(* Logix 5000 project; controller DUNEW2PLC1 vendor 1 type 14 code 221 rev 33.11; software revision 33.00; part 4 of 7 *)
(* tags used below, declared in another part *)
   BOOLS : BOOL[1024];
   DINTS : DINT[1024];
   idx_0 : DINT;
   idx_1 : DINT;
   idx_2 : DINT;
   REALS : REAL[1024];
   HomeTrigger : BOOL;
   MORE_STATS_S : BOOL[32];
   resetPB_S : BOOL;
   Safety_System_Healthy : BOOL;
   Safety_Tripped_S : BOOL;
   SegQueue : MotionSeg[32];
   X_Axis_SFX : SAFETY_FEEDBACK_INTERFACE;
   X_Axis_SLS : SAFELY_LIMITED_SPEED;
(* queued_motion, continued *)

ROUTINE MaxAbsCosSweep   (* ladder *)
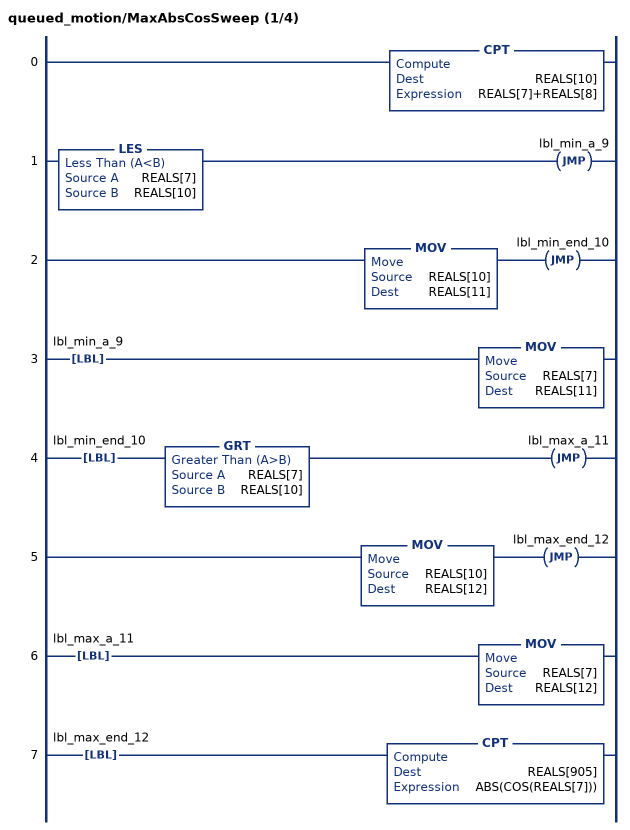
   0: CPT(REALS[10],REALS[7]+REALS[8]);
   1: LES(REALS[7],REALS[10])JMP(lbl_min_a_9);
   2: MOV(REALS[10],REALS[11])JMP(lbl_min_end_10);
   3: LBL(lbl_min_a_9)MOV(REALS[7],REALS[11]);
   4: LBL(lbl_min_end_10)GRT(REALS[7],REALS[10])JMP(lbl_max_a_11);
   5: MOV(REALS[10],REALS[12])JMP(lbl_max_end_12);
   6: LBL(lbl_max_a_11)MOV(REALS[7],REALS[12]);
   7: LBL(lbl_max_end_12)CPT(REALS[905],ABS(COS(REALS[7])));
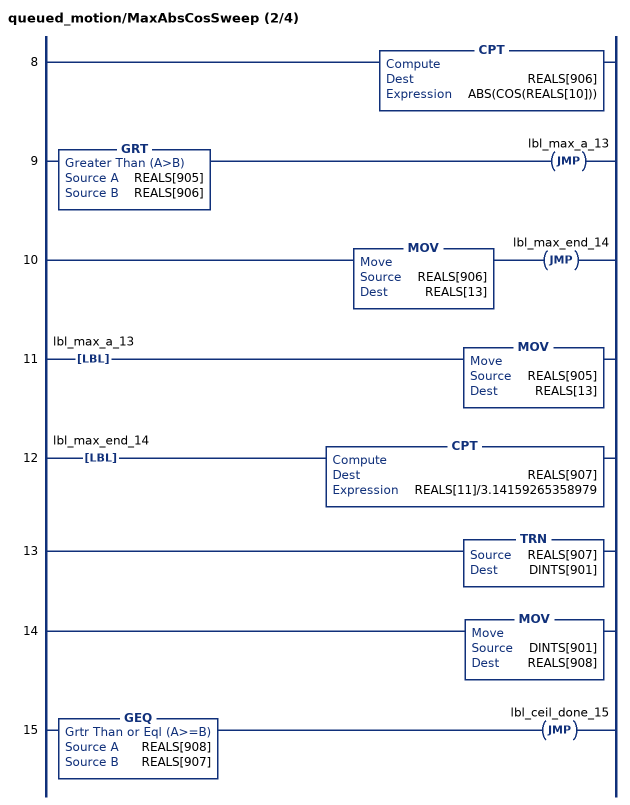
   8: CPT(REALS[906],ABS(COS(REALS[10])));
   9: GRT(REALS[905],REALS[906])JMP(lbl_max_a_13);
   10: MOV(REALS[906],REALS[13])JMP(lbl_max_end_14);
   11: LBL(lbl_max_a_13)MOV(REALS[905],REALS[13]);
   12: LBL(lbl_max_end_14)CPT(REALS[907],REALS[11]/3.14159265358979);
   13: TRN(REALS[907],DINTS[901]);
   14: MOV(DINTS[901],REALS[908]);
   15: GEQ(REALS[908],REALS[907])JMP(lbl_ceil_done_15);
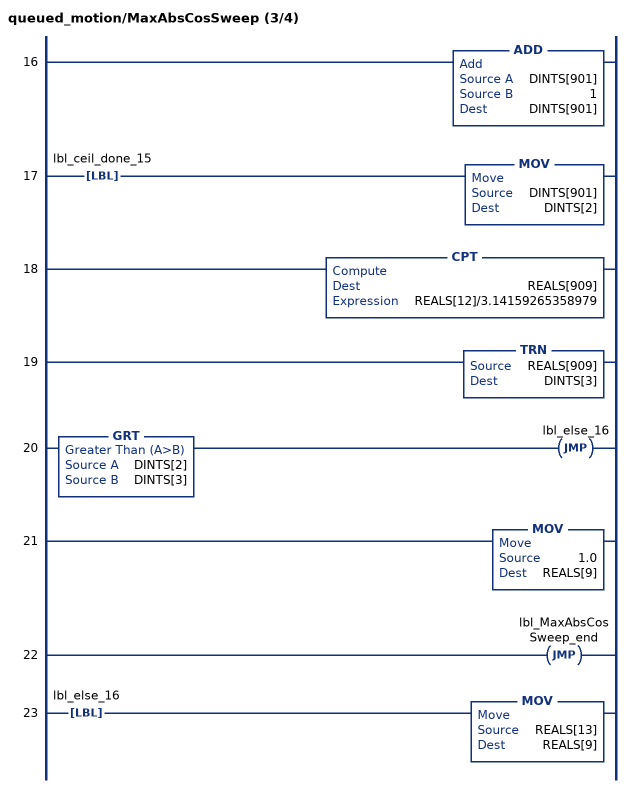
   16: ADD(DINTS[901],1,DINTS[901]);
   17: LBL(lbl_ceil_done_15)MOV(DINTS[901],DINTS[2]);
   18: CPT(REALS[909],REALS[12]/3.14159265358979);
   19: TRN(REALS[909],DINTS[3]);
   20: GRT(DINTS[2],DINTS[3])JMP(lbl_else_16);
   21: MOV(1.0,REALS[9]);
   22: JMP(lbl_MaxAbsCosSweep_end);
   23: LBL(lbl_else_16)MOV(REALS[13],REALS[9]);
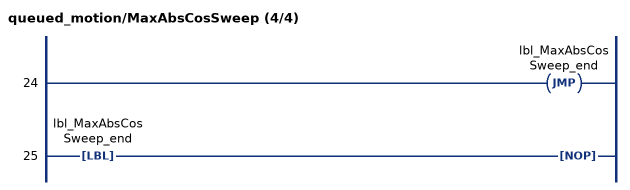
   24: JMP(lbl_MaxAbsCosSweep_end);
   25: LBL(lbl_MaxAbsCosSweep_end)NOP();
END_ROUTINE

ROUTINE MaxAbsSinSweep   (* ladder *)
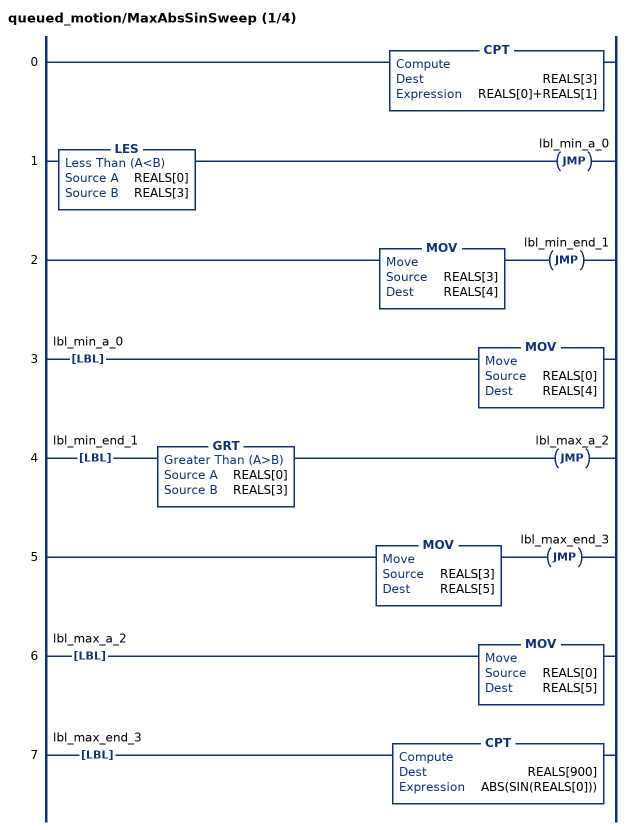
   0: CPT(REALS[3],REALS[0]+REALS[1]);
   1: LES(REALS[0],REALS[3])JMP(lbl_min_a_0);
   2: MOV(REALS[3],REALS[4])JMP(lbl_min_end_1);
   3: LBL(lbl_min_a_0)MOV(REALS[0],REALS[4]);
   4: LBL(lbl_min_end_1)GRT(REALS[0],REALS[3])JMP(lbl_max_a_2);
   5: MOV(REALS[3],REALS[5])JMP(lbl_max_end_3);
   6: LBL(lbl_max_a_2)MOV(REALS[0],REALS[5]);
   7: LBL(lbl_max_end_3)CPT(REALS[900],ABS(SIN(REALS[0])));
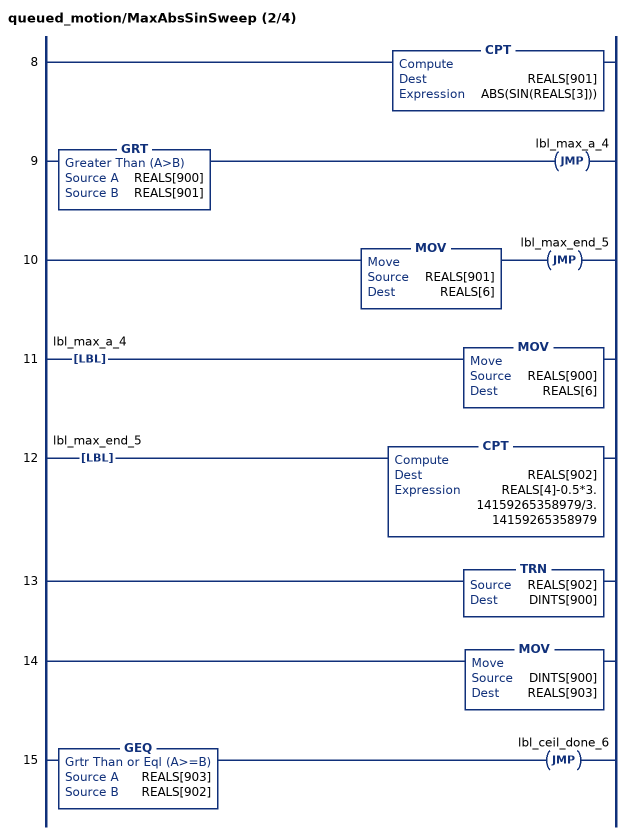
   8: CPT(REALS[901],ABS(SIN(REALS[3])));
   9: GRT(REALS[900],REALS[901])JMP(lbl_max_a_4);
   10: MOV(REALS[901],REALS[6])JMP(lbl_max_end_5);
   11: LBL(lbl_max_a_4)MOV(REALS[900],REALS[6]);
   12: LBL(lbl_max_end_5)CPT(REALS[902],REALS[4]-0.5*3.14159265358979/3.14159265358979);
   13: TRN(REALS[902],DINTS[900]);
   14: MOV(DINTS[900],REALS[903]);
   15: GEQ(REALS[903],REALS[902])JMP(lbl_ceil_done_6);
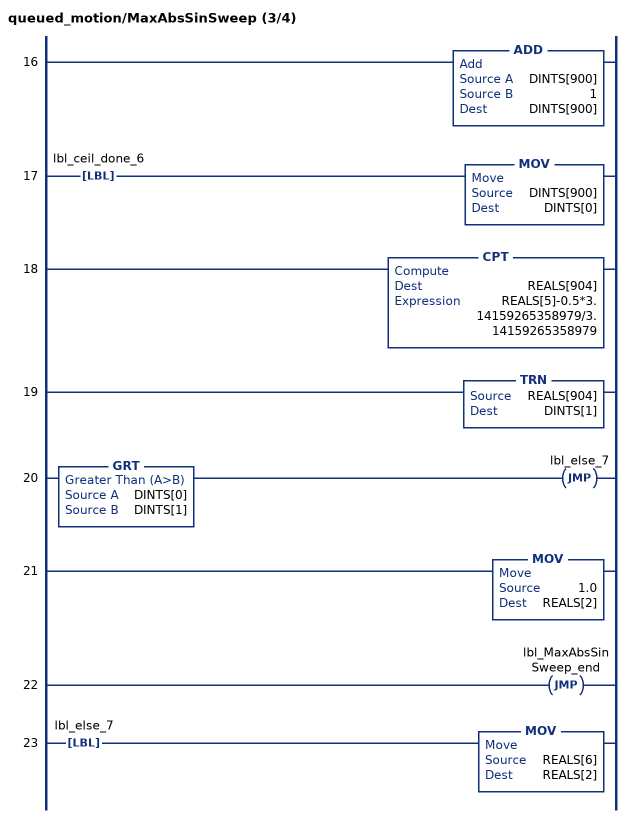
   16: ADD(DINTS[900],1,DINTS[900]);
   17: LBL(lbl_ceil_done_6)MOV(DINTS[900],DINTS[0]);
   18: CPT(REALS[904],REALS[5]-0.5*3.14159265358979/3.14159265358979);
   19: TRN(REALS[904],DINTS[1]);
   20: GRT(DINTS[0],DINTS[1])JMP(lbl_else_7);
   21: MOV(1.0,REALS[2]);
   22: JMP(lbl_MaxAbsSinSweep_end);
   23: LBL(lbl_else_7)MOV(REALS[6],REALS[2]);
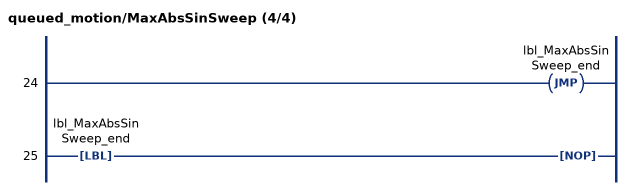
   24: JMP(lbl_MaxAbsSinSweep_end);
   25: LBL(lbl_MaxAbsSinSweep_end)NOP();
END_ROUTINE

ROUTINE SegTangentBounds   (* ladder *)
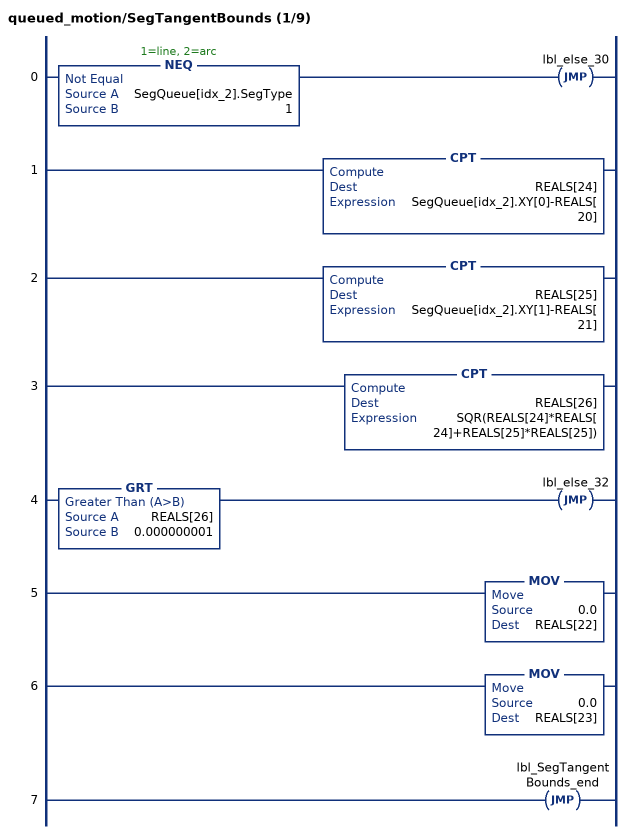
   0: NEQ(SegQueue[idx_2].SegType,1)JMP(lbl_else_30);
   1: CPT(REALS[24],SegQueue[idx_2].XY[0]-REALS[20]);
   2: CPT(REALS[25],SegQueue[idx_2].XY[1]-REALS[21]);
   3: CPT(REALS[26],SQR(REALS[24]*REALS[24]+REALS[25]*REALS[25]));
   4: GRT(REALS[26],0.000000001)JMP(lbl_else_32);
   5: MOV(0.0,REALS[22]);
   6: MOV(0.0,REALS[23]);
   7: JMP(lbl_SegTangentBounds_end);
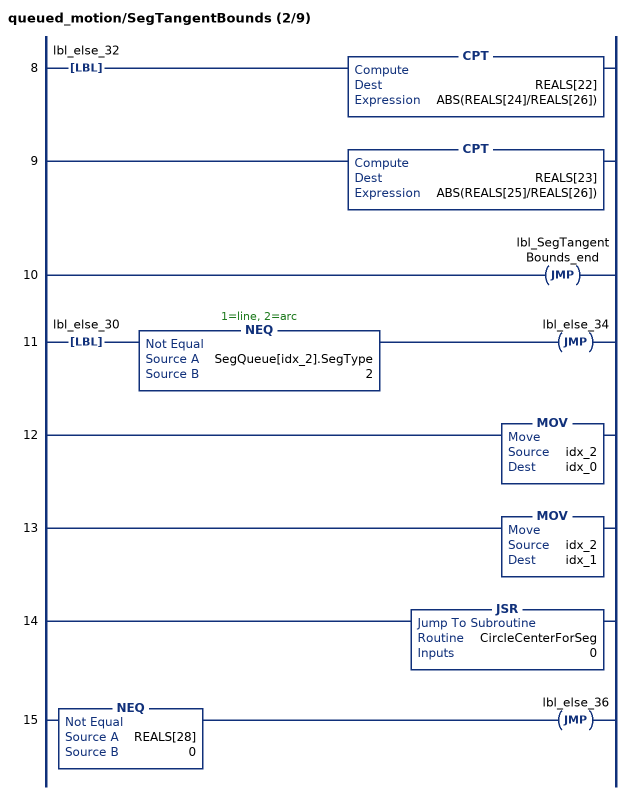
   8: LBL(lbl_else_32)CPT(REALS[22],ABS(REALS[24]/REALS[26]));
   9: CPT(REALS[23],ABS(REALS[25]/REALS[26]));
   10: JMP(lbl_SegTangentBounds_end);
   11: LBL(lbl_else_30)NEQ(SegQueue[idx_2].SegType,2)JMP(lbl_else_34);
   12: MOV(idx_2,idx_0);
   13: MOV(idx_2,idx_1);
   14: JSR(CircleCenterForSeg,0);
   15: NEQ(REALS[28],0)JMP(lbl_else_36);
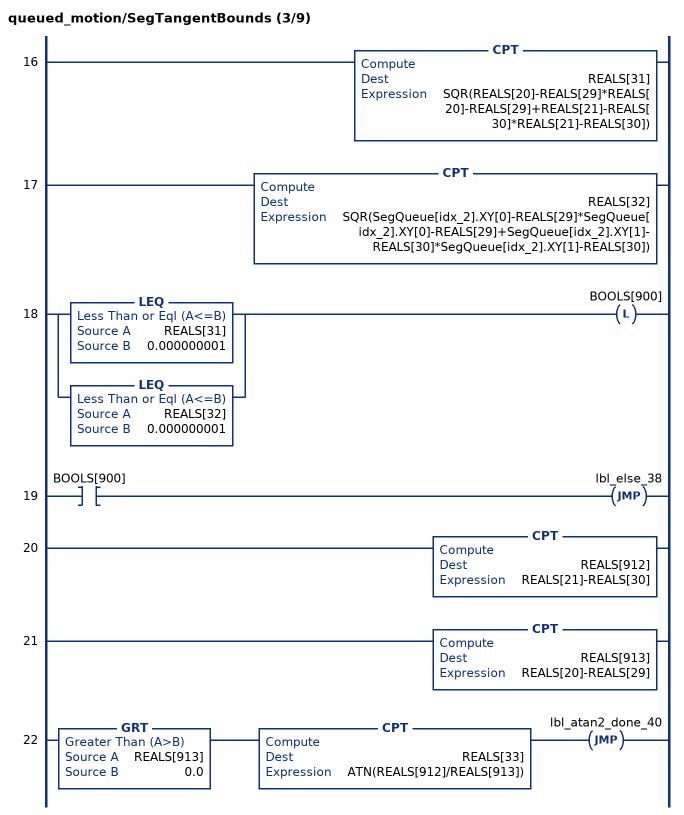
   16: CPT(REALS[31],SQR(REALS[20]-REALS[29]*REALS[20]-REALS[29]+REALS[21]-REALS[30]*REALS[21]-REALS[30]));
   17: CPT(REALS[32],SQR(SegQueue[idx_2].XY[0]-REALS[29]*SegQueue[idx_2].XY[0]-REALS[29]+SegQueue[idx_2].XY[1]-REALS[30]*SegQueue[idx_2].XY[1]-REALS[30]));
   18: [LEQ(REALS[31],0.000000001) ,LEQ(REALS[32],0.000000001) ]OTL(BOOLS[900]);
   19: XIC(BOOLS[900])JMP(lbl_else_38);
   20: CPT(REALS[912],REALS[21]-REALS[30]);
   21: CPT(REALS[913],REALS[20]-REALS[29]);
   22: GRT(REALS[913],0.0)CPT(REALS[33],ATN(REALS[912]/REALS[913]))JMP(lbl_atan2_done_40);
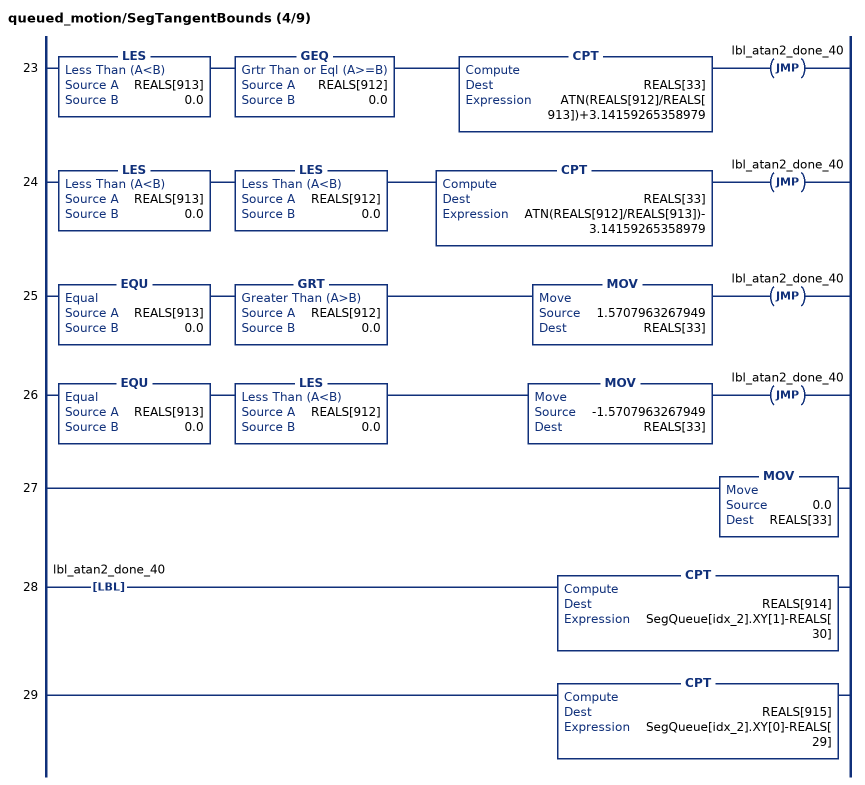
   23: LES(REALS[913],0.0)GEQ(REALS[912],0.0)CPT(REALS[33],ATN(REALS[912]/REALS[913])+3.14159265358979)JMP(lbl_atan2_done_40);
   24: LES(REALS[913],0.0)LES(REALS[912],0.0)CPT(REALS[33],ATN(REALS[912]/REALS[913])-3.14159265358979)JMP(lbl_atan2_done_40);
   25: EQU(REALS[913],0.0)GRT(REALS[912],0.0)MOV(1.5707963267949,REALS[33])JMP(lbl_atan2_done_40);
   26: EQU(REALS[913],0.0)LES(REALS[912],0.0)MOV(-1.5707963267949,REALS[33])JMP(lbl_atan2_done_40);
   27: MOV(0.0,REALS[33]);
   28: LBL(lbl_atan2_done_40)CPT(REALS[914],SegQueue[idx_2].XY[1]-REALS[30]);
   29: CPT(REALS[915],SegQueue[idx_2].XY[0]-REALS[29]);
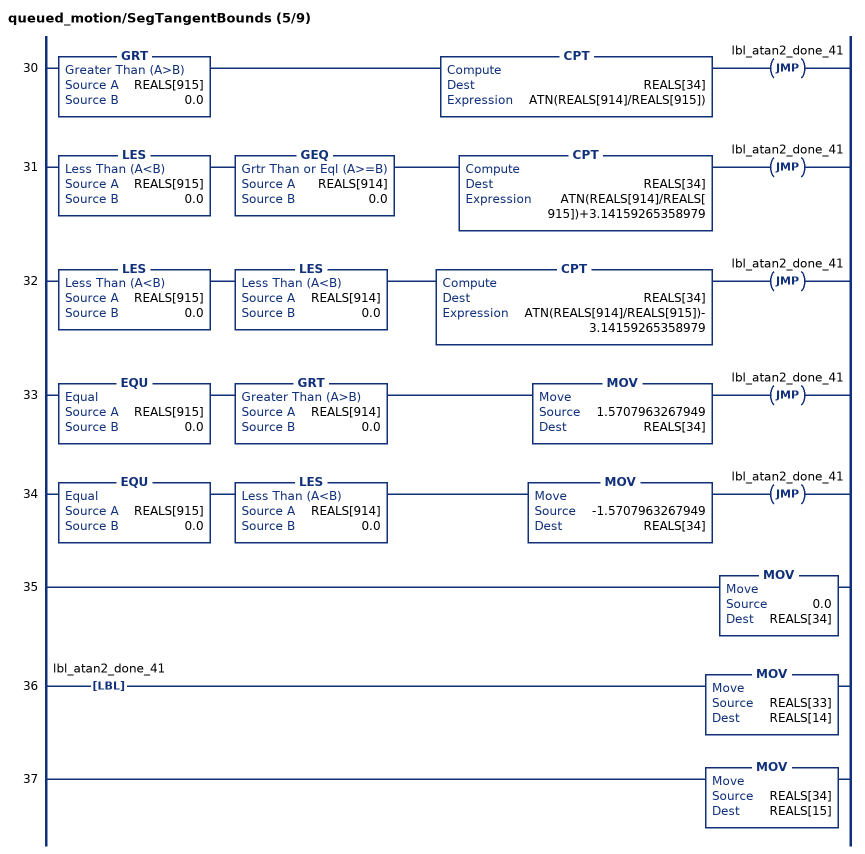
   30: GRT(REALS[915],0.0)CPT(REALS[34],ATN(REALS[914]/REALS[915]))JMP(lbl_atan2_done_41);
   31: LES(REALS[915],0.0)GEQ(REALS[914],0.0)CPT(REALS[34],ATN(REALS[914]/REALS[915])+3.14159265358979)JMP(lbl_atan2_done_41);
   32: LES(REALS[915],0.0)LES(REALS[914],0.0)CPT(REALS[34],ATN(REALS[914]/REALS[915])-3.14159265358979)JMP(lbl_atan2_done_41);
   33: EQU(REALS[915],0.0)GRT(REALS[914],0.0)MOV(1.5707963267949,REALS[34])JMP(lbl_atan2_done_41);
   34: EQU(REALS[915],0.0)LES(REALS[914],0.0)MOV(-1.5707963267949,REALS[34])JMP(lbl_atan2_done_41);
   35: MOV(0.0,REALS[34]);
   36: LBL(lbl_atan2_done_41)MOV(REALS[33],REALS[14]);
   37: MOV(REALS[34],REALS[15]);
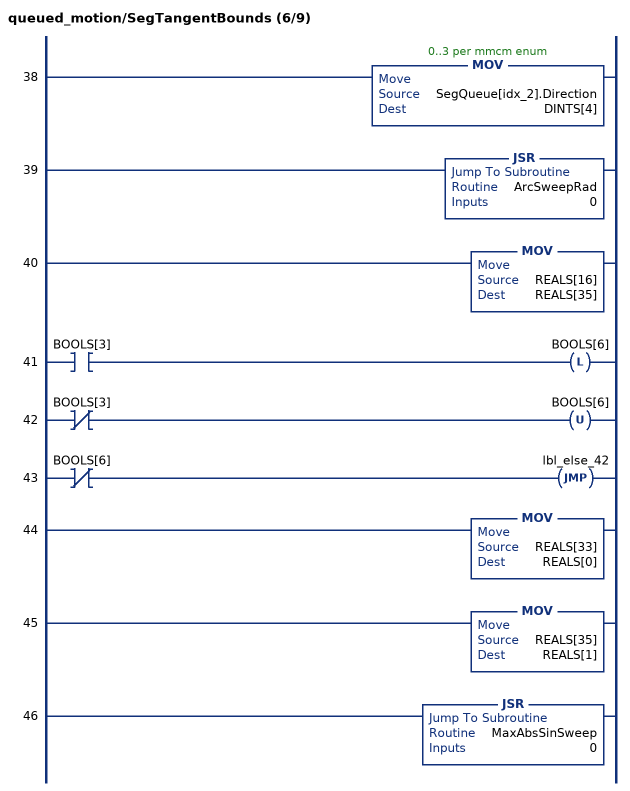
   38: MOV(SegQueue[idx_2].Direction,DINTS[4]);
   39: JSR(ArcSweepRad,0);
   40: MOV(REALS[16],REALS[35]);
   41: XIC(BOOLS[3])OTL(BOOLS[6]);
   42: XIO(BOOLS[3])OTU(BOOLS[6]);
   43: XIO(BOOLS[6])JMP(lbl_else_42);
   44: MOV(REALS[33],REALS[0]);
   45: MOV(REALS[35],REALS[1]);
   46: JSR(MaxAbsSinSweep,0);
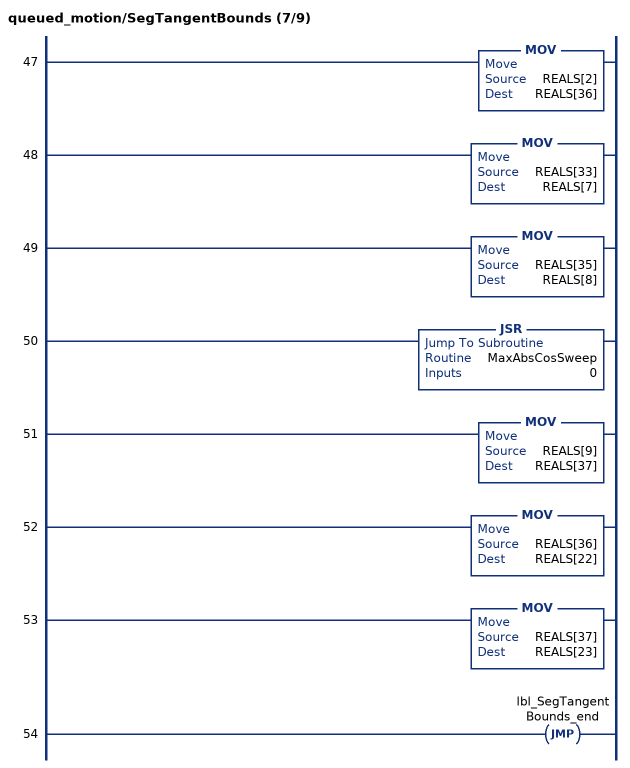
   47: MOV(REALS[2],REALS[36]);
   48: MOV(REALS[33],REALS[7]);
   49: MOV(REALS[35],REALS[8]);
   50: JSR(MaxAbsCosSweep,0);
   51: MOV(REALS[9],REALS[37]);
   52: MOV(REALS[36],REALS[22]);
   53: MOV(REALS[37],REALS[23]);
   54: JMP(lbl_SegTangentBounds_end);
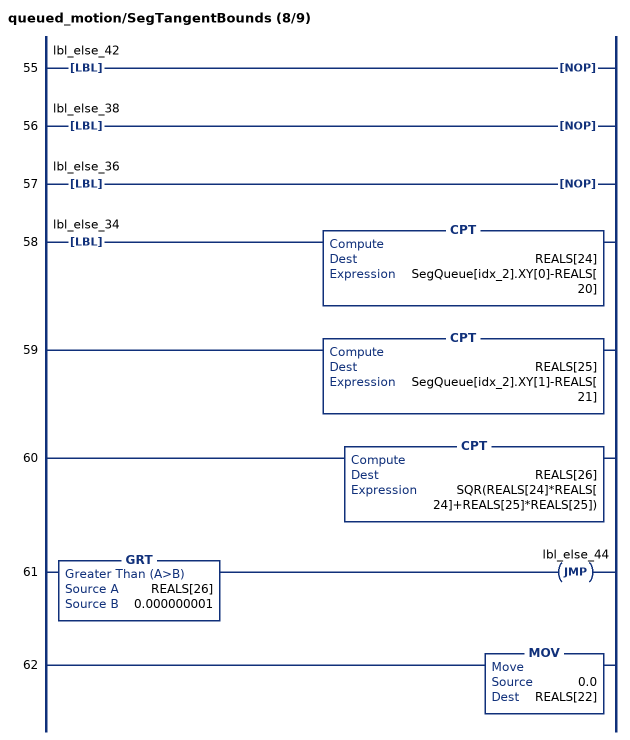
   55: LBL(lbl_else_42)NOP();
   56: LBL(lbl_else_38)NOP();
   57: LBL(lbl_else_36)NOP();
   58: LBL(lbl_else_34)CPT(REALS[24],SegQueue[idx_2].XY[0]-REALS[20]);
   59: CPT(REALS[25],SegQueue[idx_2].XY[1]-REALS[21]);
   60: CPT(REALS[26],SQR(REALS[24]*REALS[24]+REALS[25]*REALS[25]));
   61: GRT(REALS[26],0.000000001)JMP(lbl_else_44);
   62: MOV(0.0,REALS[22]);
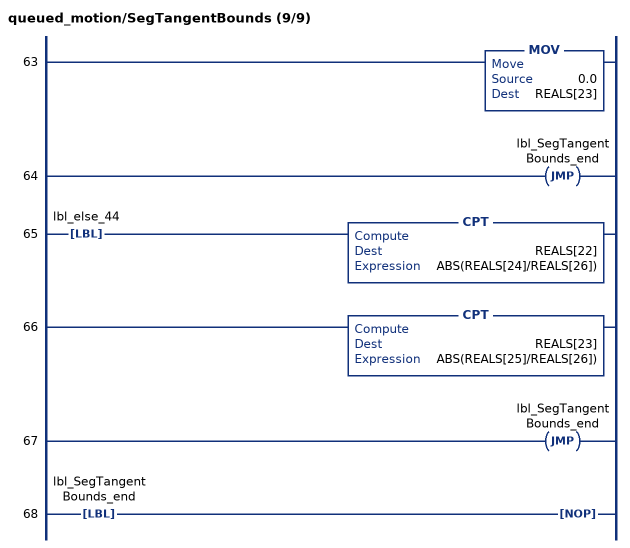
   63: MOV(0.0,REALS[23]);
   64: JMP(lbl_SegTangentBounds_end);
   65: LBL(lbl_else_44)CPT(REALS[22],ABS(REALS[24]/REALS[26]));
   66: CPT(REALS[23],ABS(REALS[25]/REALS[26]));
   67: JMP(lbl_SegTangentBounds_end);
   68: LBL(lbl_SegTangentBounds_end)NOP();
END_ROUTINE
END_PROGRAM

PROGRAM Safety   (* main routine Safety, safety *)
VAR
   e : BOOL;
   Machine_Reduced_Speed : BOOL;
END_VAR

ROUTINE Safety   (* ladder *)
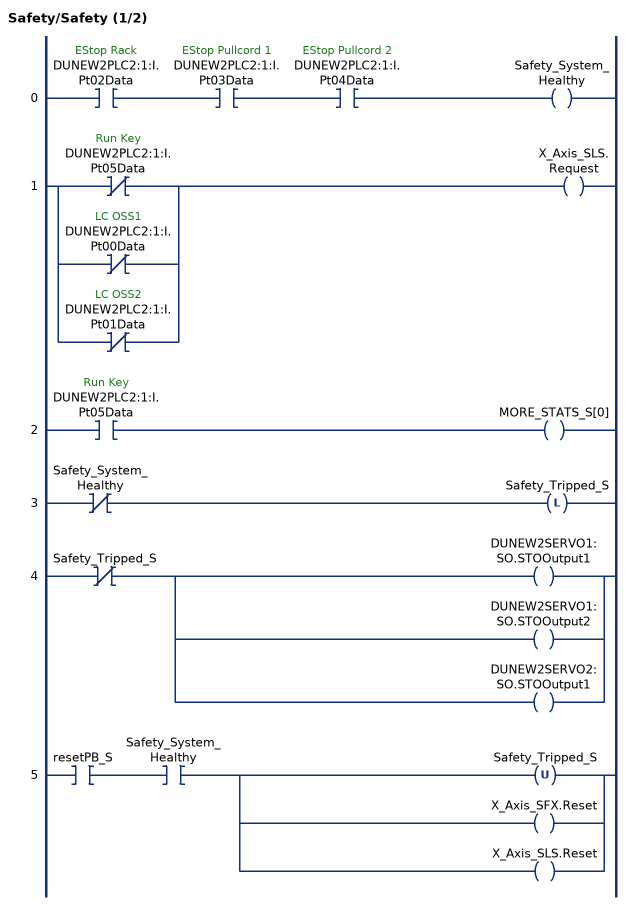
   0: XIC(DUNEW2PLC2:1:I.Pt02Data)XIC(DUNEW2PLC2:1:I.Pt03Data)XIC(DUNEW2PLC2:1:I.Pt04Data)OTE(Safety_System_Healthy);
   1: [XIO(DUNEW2PLC2:1:I.Pt05Data) ,XIO(DUNEW2PLC2:1:I.Pt00Data) ,XIO(DUNEW2PLC2:1:I.Pt01Data) ]OTE(X_Axis_SLS.Request);
   2: XIC(DUNEW2PLC2:1:I.Pt05Data)OTE(MORE_STATS_S[0]);
   3: XIO(Safety_System_Healthy)OTL(Safety_Tripped_S);
   4: XIO(Safety_Tripped_S)[[OTE(DUNEW2SERVO1:SO.STOOutput1) ,OTE(DUNEW2SERVO1:SO.STOOutput2) ] ,OTE(DUNEW2SERVO2:SO.STOOutput1) ];
   5: XIC(resetPB_S)XIC(Safety_System_Healthy)[OTU(Safety_Tripped_S) ,[OTE(X_Axis_SFX.Reset) ,OTE(X_Axis_SLS.Reset) ] ];
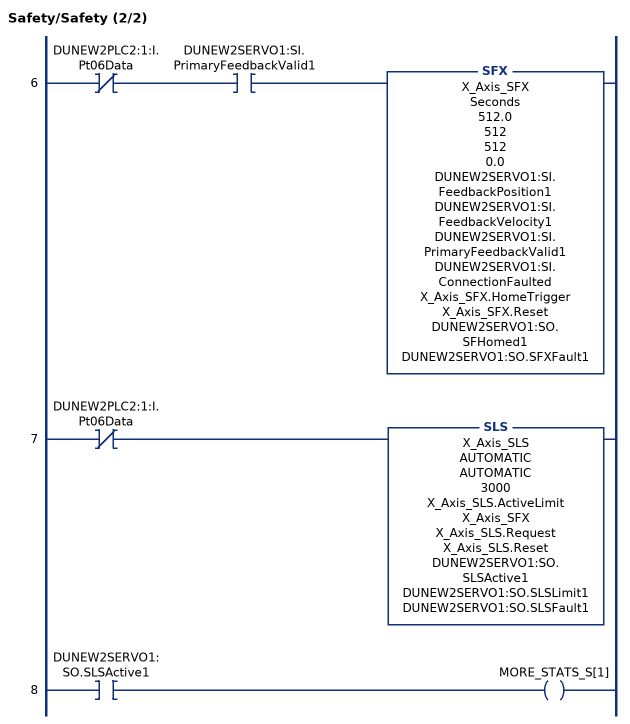
   6: XIO(DUNEW2PLC2:1:I.Pt06Data)XIC(DUNEW2SERVO1:SI.PrimaryFeedbackValid1)SFX(X_Axis_SFX,Seconds,512.0,512,512,0.0,DUNEW2SERVO1:SI.FeedbackPosition1,DUNEW2SERVO1:SI.FeedbackVelocity1,DUNEW2SERVO1:SI.PrimaryFeedbackValid1,DUNEW2SERVO1:SI.ConnectionFaulted,X_Axis_SFX.HomeTrigger,X_Axis_SFX.Reset,DUNEW2SERVO1:SO.SFHomed1,DUNEW2SERVO1:SO.SFXFault1);
   7: XIO(DUNEW2PLC2:1:I.Pt06Data)SLS(X_Axis_SLS,AUTOMATIC,AUTOMATIC,3000,X_Axis_SLS.ActiveLimit,X_Axis_SFX,X_Axis_SLS.Request,X_Axis_SLS.Reset,DUNEW2SERVO1:SO.SLSActive1,DUNEW2SERVO1:SO.SLSLimit1,DUNEW2SERVO1:SO.SLSFault1);
   8: XIC(DUNEW2SERVO1:SO.SLSActive1)OTE(MORE_STATS_S[1]);
END_ROUTINE
END_PROGRAM
